SUBAPPLICATION Uebung_022 (* Subapplication Type *)
  (* Standard: 61499-2 *)
  (* Version 1.0, 2023-10-23, franz *)
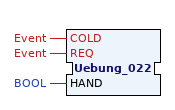
  EVENT_INPUT
    COLD;
    REQ;
  END_EVENT
  VAR_INPUT
    HAND : BOOL;
  END_VAR
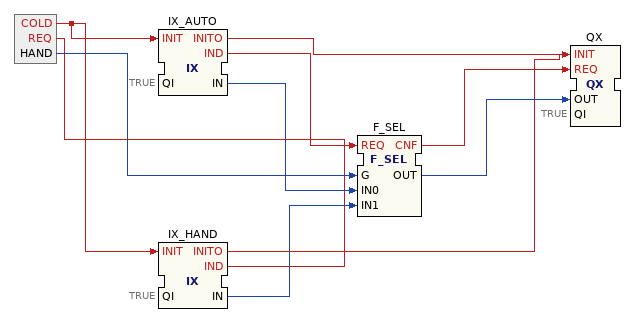
  FBS
    QX : QX(QI := TRUE);
    IX_AUTO : IX(QI := TRUE);
    IX_HAND : IX(QI := TRUE);
    F_SEL : F_SEL;
  END_FBS
  EVENT_CONNECTIONS
    COLD TO IX_AUTO.INIT;
    IX_AUTO.INITO TO QX.INIT;
    COLD TO IX_HAND.INIT;
    IX_HAND.INITO TO QX.INIT;
    F_SEL.CNF TO QX.REQ;
    IX_AUTO.IND TO F_SEL.REQ;
    IX_HAND.IND TO F_SEL.REQ;
    REQ TO F_SEL.REQ;
  END_CONNECTIONS
  DATA_CONNECTIONS
    HAND TO F_SEL.G;
    IX_AUTO.IN TO F_SEL.IN0;
    IX_HAND.IN TO F_SEL.IN1;
    F_SEL.OUT TO QX.OUT;
  END_CONNECTIONS
END_SUBAPPLICATION
